TYPE ZDataMachine :
STRUCT
{region "PrimaryGear"}
{IF NOT (defined (PrimaryGear_disabled))}
  PrimaryGear : GearDataMachine;
  {attribute 'ZId' := 'd1deea68-6f8b-4ea5-9916-7be69dc951fa'}
{END_IF}
{endregion}
{region "Machine"}
{IF NOT (defined (Machine_disabled))}
  Machine : MachineDataMachine;
  {attribute 'ZId' := '9a1e8940-043c-4b8f-bd95-526fb267b71c'}
{END_IF}
{endregion}
{region "SimpleGear"}
{IF NOT (defined (SimpleGear_disabled))}
  SimpleGear : GearDataMachine;
  {attribute 'ZId' := '215d1db4-d61a-4f46-91b5-612373b86c91'}
{END_IF}
{endregion}
{region "StruckigGear"}
{IF NOT (defined (StruckigGear_disabled))}
  StruckigGear : GearDataMachine;
  {attribute 'ZId' := 'd827270e-999f-436d-80d5-b12442f5d1cf'}
{END_IF}
{endregion}
{attribute '__ZwPlcApplicationDataMachineDeclaration__'} // Do not remove this attribute! It is used for code generation.
END_STRUCT
END_TYPE

(* stored: Version 1.1.0.1
   DUT ZDataMachine: Id {02091abb-4abd-4a25-9b25-cb7938611ab5} *)
